// Mitsubishi GX Developer project: 20100302伺服締付機V02   PLC: FX3G

PROGRAM MAIN
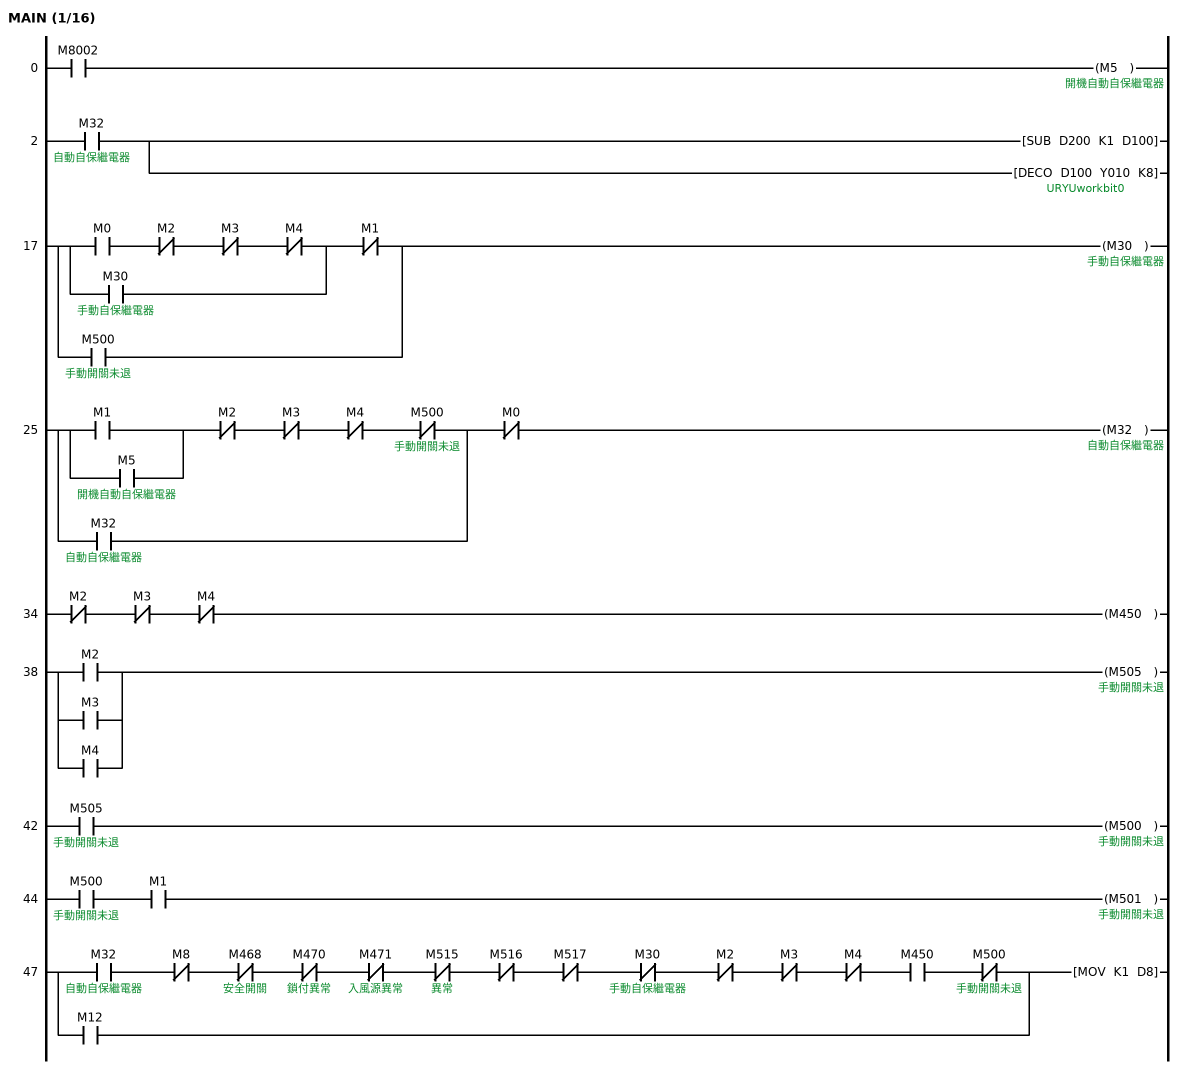
0     LD      M8002
      OUT     M5  ; 開機自動自保繼電器
2     LD      M32  ; 自動自保繼電器
      SUB     D200 K1 D100
        [note] 模組選擇
      DECO    D100 Y010 K8  ; URYUworkbit0
17    LD      M0
      ANI     M2
      ANI     M3
      ANI     M4
      OR      M30  ; 手動自保繼電器
      ANI     M1
      OR      M500  ; 手動開關未退
      OUT     M30  ; 手動自保繼電器
25    LD      M1
      OR      M5  ; 開機自動自保繼電器
      ANI     M2
      ANI     M3
      ANI     M4
      ANI     M500  ; 手動開關未退
      OR      M32  ; 自動自保繼電器
      ANI     M0
      OUT     M32  ; 自動自保繼電器
34    LDI     M2
      ANI     M3
      ANI     M4
      OUT     M450
38    LD      M2
      OR      M3
      OR      M4
      OUT     M505  ; 手動開關未退
42    LD      M505  ; 手動開關未退
      OUT     M500  ; 手動開關未退
44    LD      M500  ; 手動開關未退
      AND     M1
      OUT     M501  ; 手動開關未退
47    LD      M32  ; 自動自保繼電器
      ANI     M8
      ANI     M468  ; 安全開關
      ANI     M470  ; 鎖付異常
      ANI     M471  ; 入風源異常
      ANI     M515  ; 異常
      ANI     M516
      ANI     M517
      ANI     M30  ; 手動自保繼電器
      ANI     M2
      ANI     M3
      ANI     M4
      AND     M450
      ANI     M500  ; 手動開關未退
      OR      M12
      MOV     K1 D8
        [note] 自動畫面
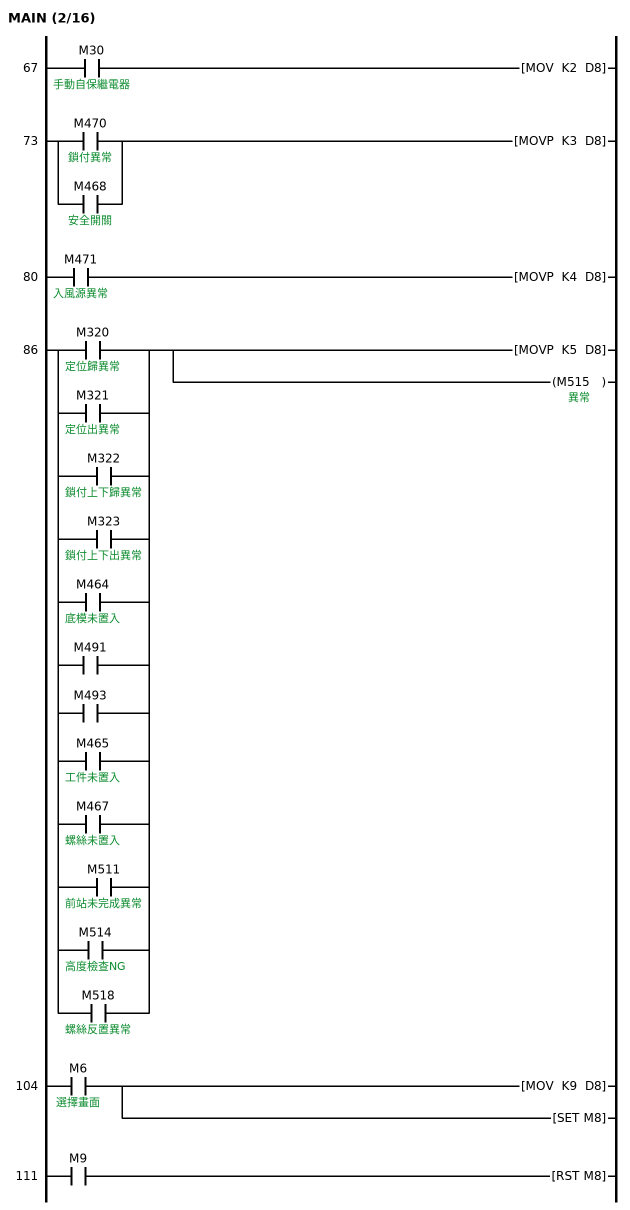
67    LD      M30  ; 手動自保繼電器
      MOV     K2 D8
        [note] 手動畫面
73    LD      M470  ; 鎖付異常
      OR      M468  ; 安全開關
      MOVP    K3 D8
        [note] 異常畫面
80    LD      M471  ; 入風源異常
      MOVP    K4 D8
        [note] 入風源異常畫面
86    LD      M320  ; 定位歸異常
      OR      M321  ; 定位出異常
      OR      M322  ; 鎖付上下歸異常
      OR      M323  ; 鎖付上下出異常
      OR      M464  ; 底模未置入
      OR      M491
      OR      M493
      OR      M465  ; 工件未置入
      OR      M467  ; 螺絲未置入
      OR      M511  ; 前站未完成異常
      OR      M514  ; 高度檢查NG
      OR      M518  ; 螺絲反置異常
      MOVP    K5 D8
        [note] 磁簧開關異常畫面
      OUT     M515  ; 異常
104   LD      M6  ; 選擇畫面
      MOV     K9 D8
      SET     M8
111   LD      M9
      RST     M8
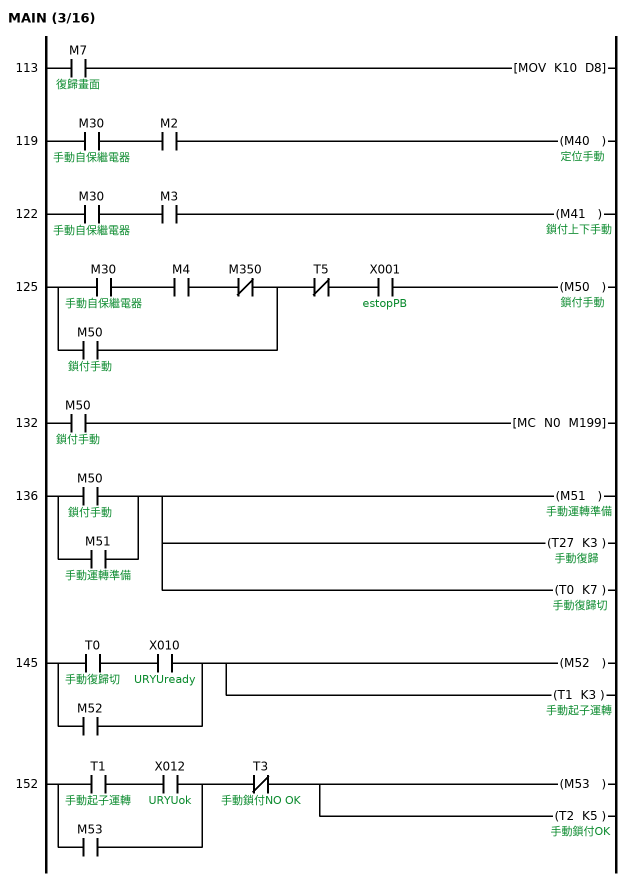
113   LD      M7  ; 復歸畫面
      MOV     K10 D8
119   LD      M30  ; 手動自保繼電器
      AND     M2
      OUT     M40  ; 定位手動
122   LD      M30  ; 手動自保繼電器
      AND     M3
      OUT     M41  ; 鎖付上下手動
125   LD      M30  ; 手動自保繼電器
      AND     M4
      ANI     M350
      OR      M50  ; 鎖付手動
      ANI     T5
      AND     X001  ; estopPB
      OUT     M50  ; 鎖付手動
132   LD      M50  ; 鎖付手動
      MC      N0 M199
136   LD      M50  ; 鎖付手動
      OR      M51  ; 手動運轉準備
      OUT     M51  ; 手動運轉準備
      OUT     T27 K3  ; 手動復歸
      OUT     T0 K7  ; 手動復歸切
145   LD      T0  ; 手動復歸切
      AND     X010  ; URYUready
      OR      M52
      OUT     M52
      OUT     T1 K3  ; 手動起子運轉
152   LD      T1  ; 手動起子運轉
      AND     X012  ; URYUok
      OR      M53
      ANI     T3  ; 手動鎖付NO OK
      OUT     M53
      OUT     T2 K5  ; 手動鎖付OK
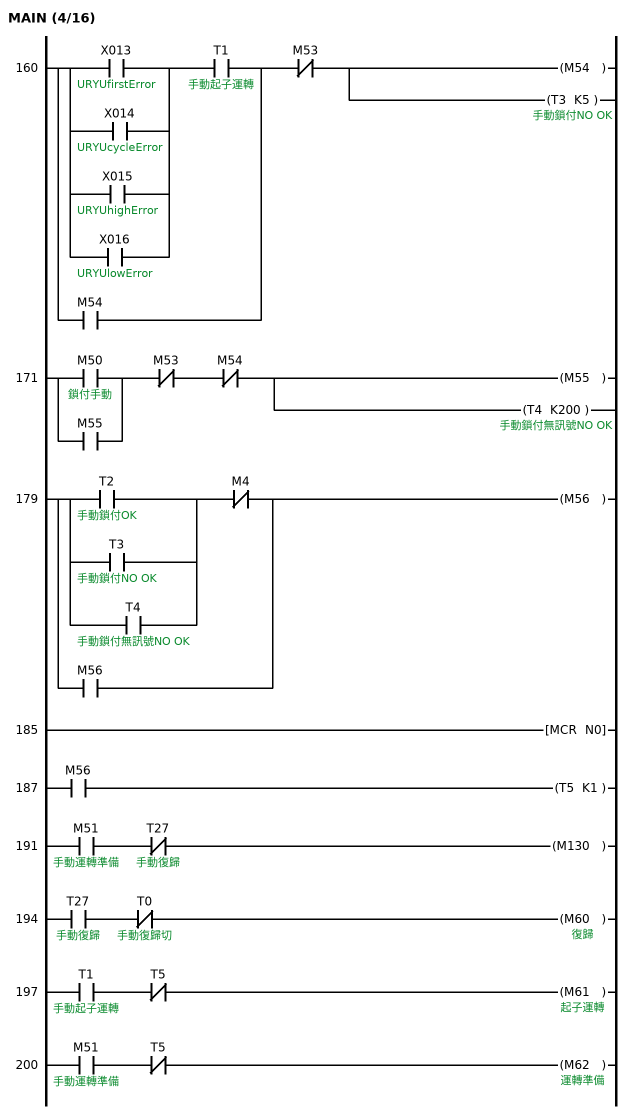
160   LD      X013  ; URYUfirstError
      OR      X014  ; URYUcycleError
      OR      X015  ; URYUhighError
      OR      X016  ; URYUlowError
      AND     T1  ; 手動起子運轉
      OR      M54
      ANI     M53
      OUT     M54
      OUT     T3 K5  ; 手動鎖付NO OK
171   LD      M50  ; 鎖付手動
      OR      M55
      ANI     M53
      ANI     M54
      OUT     M55
      OUT     T4 K200  ; 手動鎖付無訊號NO OK
179   LD      T2  ; 手動鎖付OK
      OR      T3  ; 手動鎖付NO OK
      OR      T4  ; 手動鎖付無訊號NO OK
      ANI     M4
      OR      M56
      OUT     M56
185   MCR     N0
187   LD      M56
      OUT     T5 K1
191   LD      M51  ; 手動運轉準備
      ANI     T27  ; 手動復歸
      OUT     M130
194   LD      T27  ; 手動復歸
      ANI     T0  ; 手動復歸切
      OUT     M60  ; 復歸
197   LD      T1  ; 手動起子運轉
      ANI     T5
      OUT     M61  ; 起子運轉
200   LD      M51  ; 手動運轉準備
      ANI     T5
      OUT     M62  ; 運轉準備
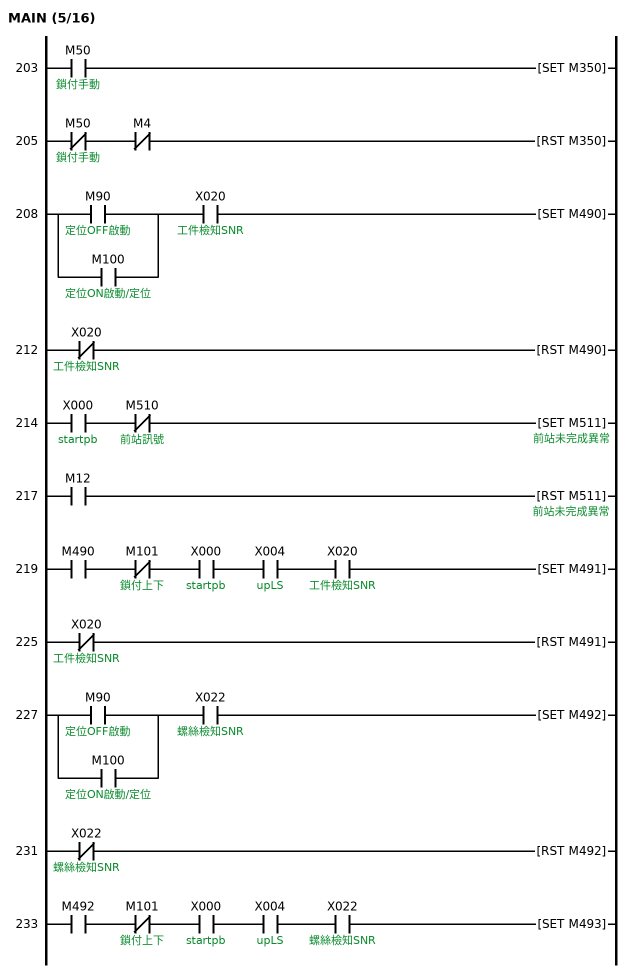
203   LD      M50  ; 鎖付手動
      SET     M350
205   LDI     M50  ; 鎖付手動
      ANI     M4
      RST     M350
208   LD      M90  ; 定位OFF啟動
      OR      M100  ; 定位ON啟動/定位
      AND     X020  ; 工件檢知SNR
      SET     M490
212   LDI     X020  ; 工件檢知SNR
      RST     M490
214   LD      X000  ; startpb
      ANI     M510  ; 前站訊號
      SET     M511  ; 前站未完成異常
217   LD      M12
      RST     M511  ; 前站未完成異常
219   LD      M490
      ANI     M101  ; 鎖付上下
      AND     X000  ; startpb
      AND     X004  ; upLS
      AND     X020  ; 工件檢知SNR
      SET     M491
225   LDI     X020  ; 工件檢知SNR
      RST     M491
227   LD      M90  ; 定位OFF啟動
      OR      M100  ; 定位ON啟動/定位
      AND     X022  ; 螺絲檢知SNR
      SET     M492
231   LDI     X022  ; 螺絲檢知SNR
      RST     M492
233   LD      M492
      ANI     M101  ; 鎖付上下
      AND     X000  ; startpb
      AND     X004  ; upLS
      AND     X022  ; 螺絲檢知SNR
      SET     M493
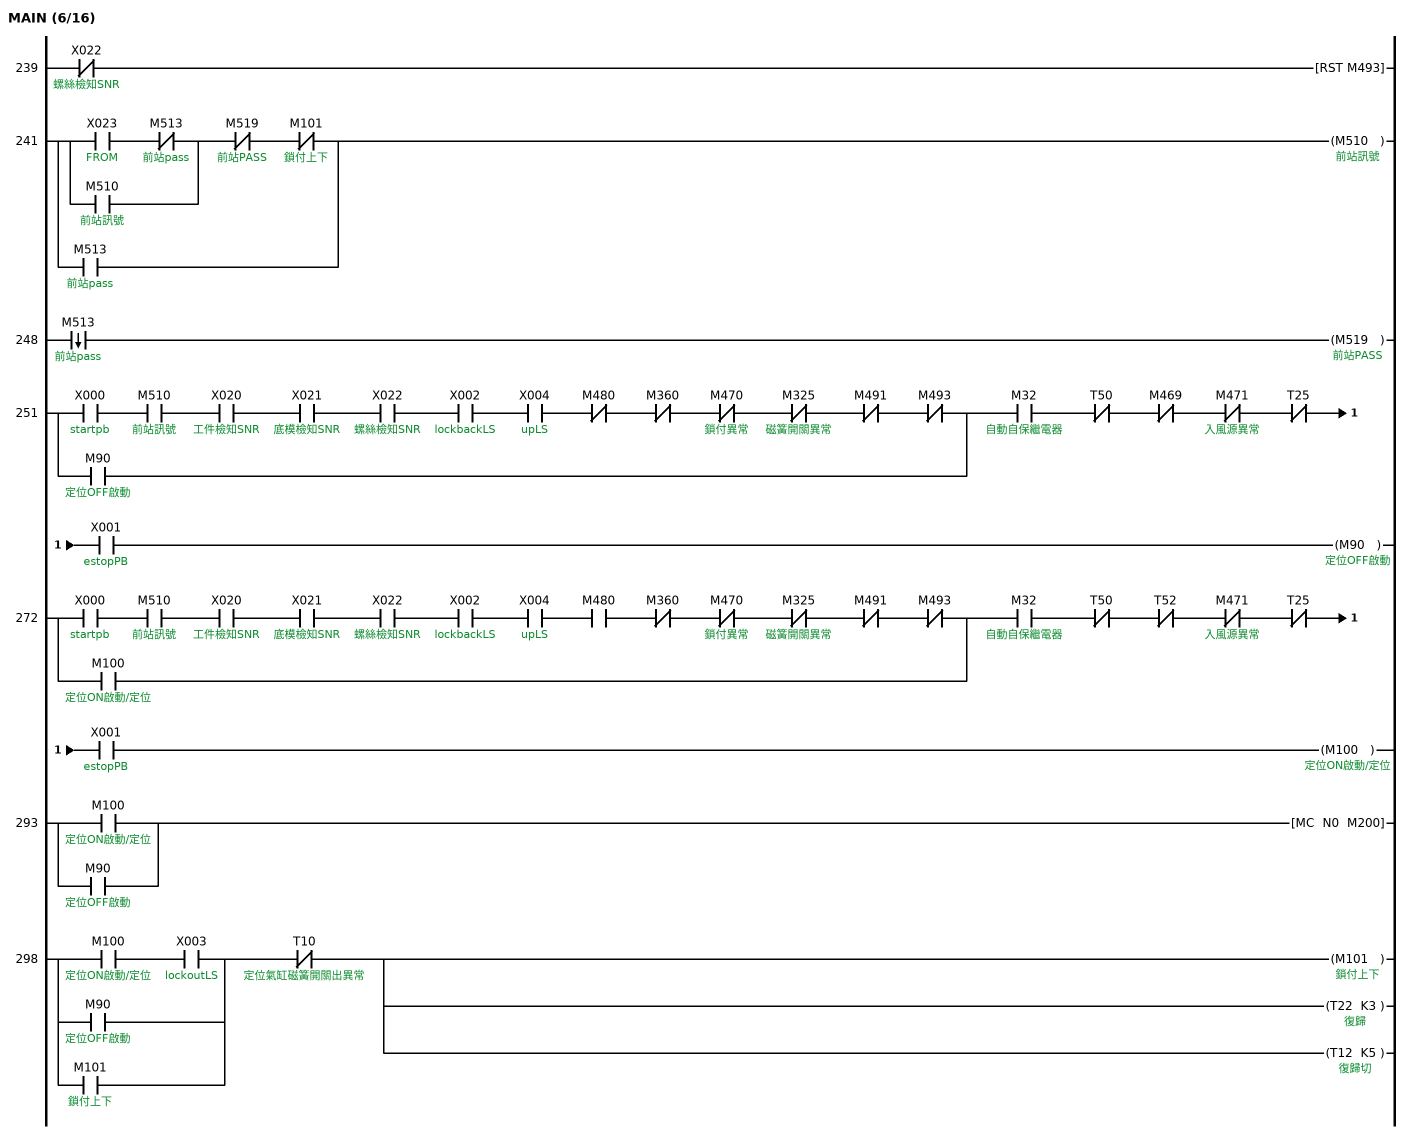
239   LDI     X022  ; 螺絲檢知SNR
      RST     M493
241   LD      X023  ; FROM
      ANI     M513  ; 前站pass
      OR      M510  ; 前站訊號
      ANI     M519  ; 前站PASS
      ANI     M101  ; 鎖付上下
      OR      M513  ; 前站pass
      OUT     M510  ; 前站訊號
248   LDF     M513  ; 前站pass
      OUT     M519  ; 前站PASS
251   LD      X000  ; startpb
      AND     M510  ; 前站訊號
      AND     X020  ; 工件檢知SNR
      AND     X021  ; 底模檢知SNR
      AND     X022  ; 螺絲檢知SNR
      AND     X002  ; lockbackLS
      AND     X004  ; upLS
      ANI     M480
      ANI     M360
      ANI     M470  ; 鎖付異常
      ANI     M325  ; 磁簧開關異常
      ANI     M491
      ANI     M493
      OR      M90  ; 定位OFF啟動
      AND     M32  ; 自動自保繼電器
      ANI     T50
      ANI     M469
      ANI     M471  ; 入風源異常
      ANI     T25
      AND     X001  ; estopPB
      OUT     M90  ; 定位OFF啟動
272   LD      X000  ; startpb
      AND     M510  ; 前站訊號
      AND     X020  ; 工件檢知SNR
      AND     X021  ; 底模檢知SNR
      AND     X022  ; 螺絲檢知SNR
      AND     X002  ; lockbackLS
      AND     X004  ; upLS
      AND     M480
      ANI     M360
      ANI     M470  ; 鎖付異常
      ANI     M325  ; 磁簧開關異常
      ANI     M491
      ANI     M493
      OR      M100  ; 定位ON啟動/定位
      AND     M32  ; 自動自保繼電器
      ANI     T50
      ANI     T52
      ANI     M471  ; 入風源異常
      ANI     T25
      AND     X001  ; estopPB
      OUT     M100  ; 定位ON啟動/定位
293   LD      M100  ; 定位ON啟動/定位
      OR      M90  ; 定位OFF啟動
      MC      N0 M200
298   LD      M100  ; 定位ON啟動/定位
      AND     X003  ; lockoutLS
      OR      M90  ; 定位OFF啟動
      OR      M101  ; 鎖付上下
      ANI     T10  ; 定位氣缸磁簧開關出異常
      OUT     M101  ; 鎖付上下
      OUT     T22 K3  ; 復歸
      OUT     T12 K5  ; 復歸切
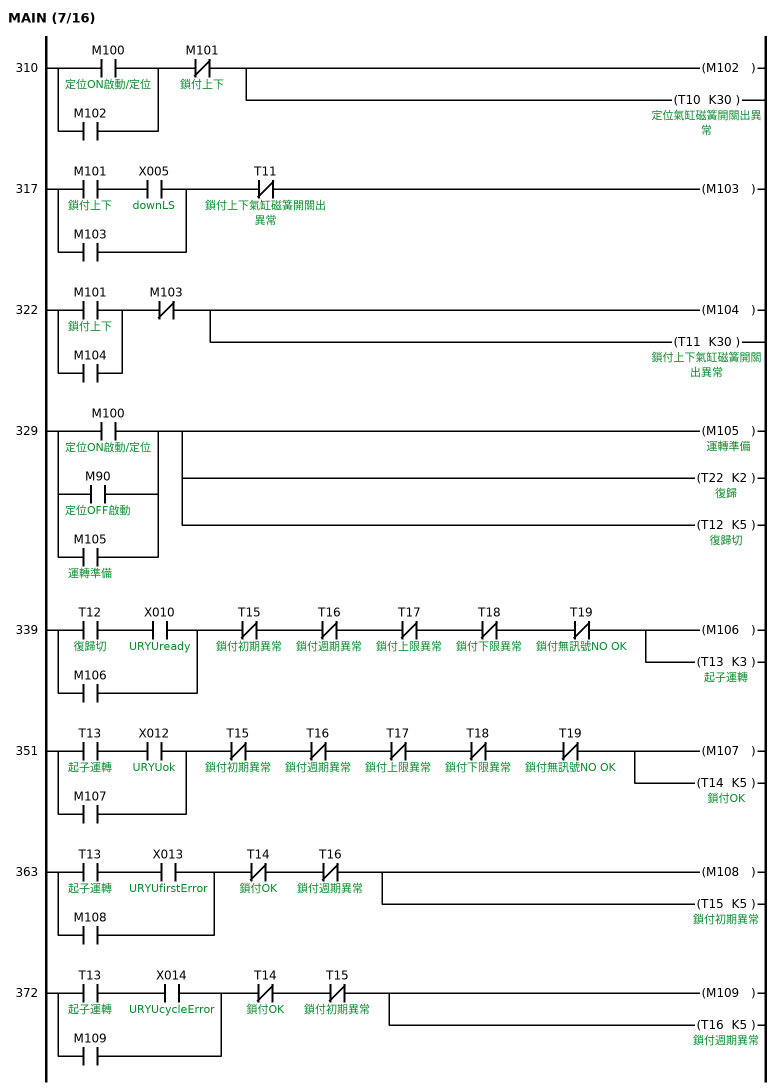
310   LD      M100  ; 定位ON啟動/定位
      OR      M102
      ANI     M101  ; 鎖付上下
      OUT     M102
      OUT     T10 K30  ; 定位氣缸磁簧開關出異常
317   LD      M101  ; 鎖付上下
      AND     X005  ; downLS
      OR      M103
      ANI     T11  ; 鎖付上下氣缸磁簧開關出異常
      OUT     M103
322   LD      M101  ; 鎖付上下
      OR      M104
      ANI     M103
      OUT     M104
      OUT     T11 K30  ; 鎖付上下氣缸磁簧開關出異常
329   LD      M100  ; 定位ON啟動/定位
      OR      M90  ; 定位OFF啟動
      OR      M105  ; 運轉準備
      OUT     M105  ; 運轉準備
      OUT     T22 K2  ; 復歸
      OUT     T12 K5  ; 復歸切
339   LD      T12  ; 復歸切
      AND     X010  ; URYUready
      OR      M106
      ANI     T15  ; 鎖付初期異常
      ANI     T16  ; 鎖付週期異常
      ANI     T17  ; 鎖付上限異常
      ANI     T18  ; 鎖付下限異常
      ANI     T19  ; 鎖付無訊號NO OK
      OUT     M106
      OUT     T13 K3  ; 起子運轉
351   LD      T13  ; 起子運轉
      AND     X012  ; URYUok
      OR      M107
      ANI     T15  ; 鎖付初期異常
      ANI     T16  ; 鎖付週期異常
      ANI     T17  ; 鎖付上限異常
      ANI     T18  ; 鎖付下限異常
      ANI     T19  ; 鎖付無訊號NO OK
      OUT     M107
      OUT     T14 K5  ; 鎖付OK
363   LD      T13  ; 起子運轉
      AND     X013  ; URYUfirstError
      OR      M108
      ANI     T14  ; 鎖付OK
      ANI     T16  ; 鎖付週期異常
      OUT     M108
      OUT     T15 K5  ; 鎖付初期異常
372   LD      T13  ; 起子運轉
      AND     X014  ; URYUcycleError
      OR      M109
      ANI     T14  ; 鎖付OK
      ANI     T15  ; 鎖付初期異常
      OUT     M109
      OUT     T16 K5  ; 鎖付週期異常
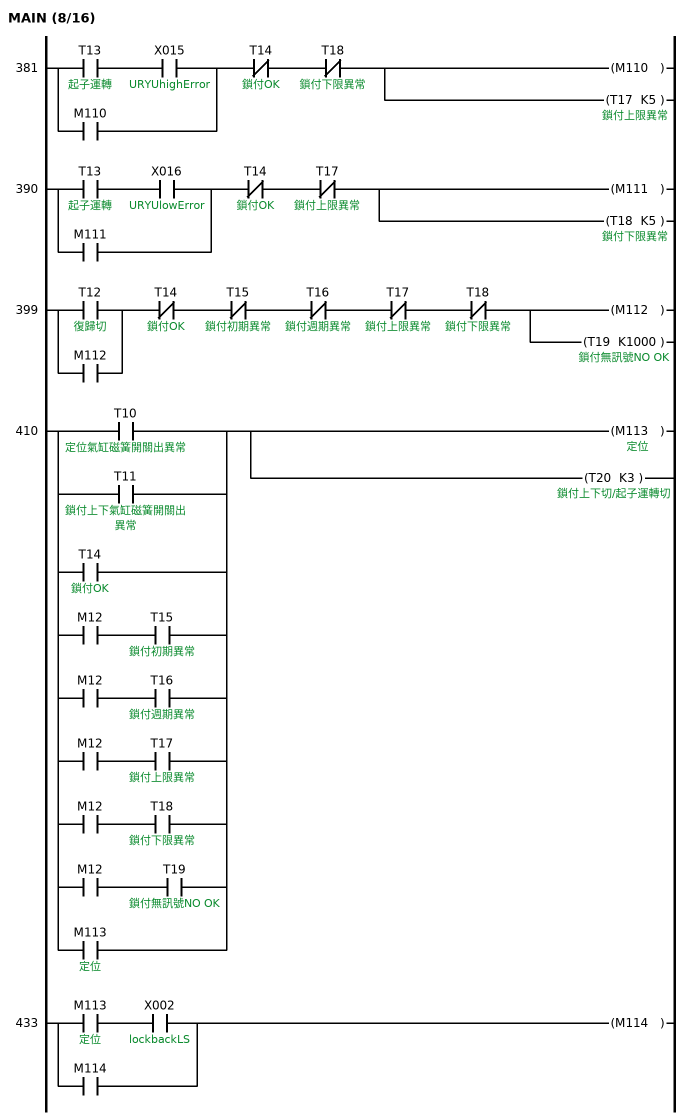
381   LD      T13  ; 起子運轉
      AND     X015  ; URYUhighError
      OR      M110
      ANI     T14  ; 鎖付OK
      ANI     T18  ; 鎖付下限異常
      OUT     M110
      OUT     T17 K5  ; 鎖付上限異常
390   LD      T13  ; 起子運轉
      AND     X016  ; URYUlowError
      OR      M111
      ANI     T14  ; 鎖付OK
      ANI     T17  ; 鎖付上限異常
      OUT     M111
      OUT     T18 K5  ; 鎖付下限異常
399   LD      T12  ; 復歸切
      OR      M112
      ANI     T14  ; 鎖付OK
      ANI     T15  ; 鎖付初期異常
      ANI     T16  ; 鎖付週期異常
      ANI     T17  ; 鎖付上限異常
      ANI     T18  ; 鎖付下限異常
      OUT     M112
      OUT     T19 K1000  ; 鎖付無訊號NO OK
410   LD      T10  ; 定位氣缸磁簧開關出異常
      OR      T11  ; 鎖付上下氣缸磁簧開關出異常
      OR      T14  ; 鎖付OK
      LD      M12
      AND     T15  ; 鎖付初期異常
      ORB
      LD      M12
      AND     T16  ; 鎖付週期異常
      ORB
      LD      M12
      AND     T17  ; 鎖付上限異常
      ORB
      LD      M12
      AND     T18  ; 鎖付下限異常
      ORB
      LD      M12
      AND     T19  ; 鎖付無訊號NO OK
      ORB
      OR      M113  ; 定位
      OUT     M113  ; 定位
      OUT     T20 K3  ; 鎖付上下切/起子運轉切
433   LD      M113  ; 定位
      AND     X002  ; lockbackLS
      OR      M114
      OUT     M114
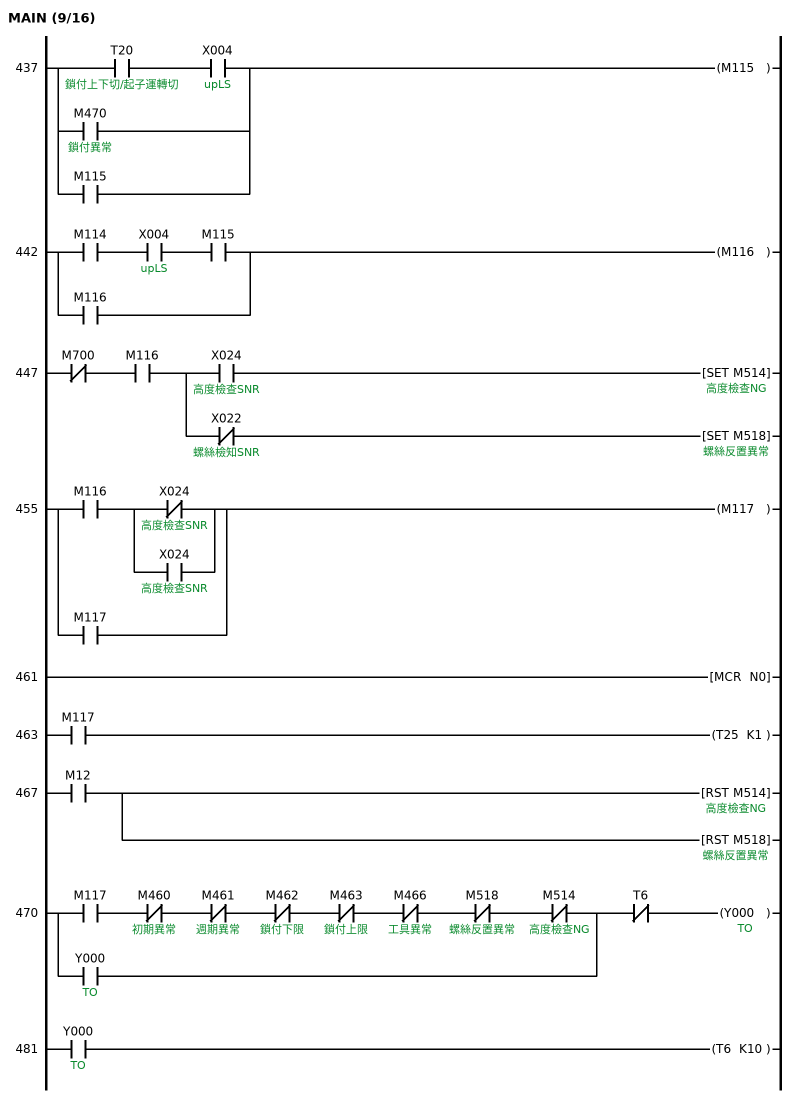
437   LD      T20  ; 鎖付上下切/起子運轉切
      AND     X004  ; upLS
      OR      M470  ; 鎖付異常
      OR      M115
      OUT     M115
442   LD      M114
      AND     X004  ; upLS
      AND     M115
      OR      M116
      OUT     M116
447   LDI     M700
      AND     M116
      MPS
      AND     X024  ; 高度檢查SNR
      SET     M514  ; 高度檢查NG
      MPP
      ANI     X022  ; 螺絲檢知SNR
      SET     M518  ; 螺絲反置異常
455   LD      M116
      LDI     X024  ; 高度檢查SNR
      OR      X024  ; 高度檢查SNR
      ANB
      OR      M117
      OUT     M117
461   MCR     N0
463   LD      M117
      OUT     T25 K1
467   LD      M12
      RST     M514  ; 高度檢查NG
      RST     M518  ; 螺絲反置異常
470   LD      M117
      ANI     M460  ; 初期異常
      ANI     M461  ; 週期異常
      ANI     M462  ; 鎖付下限
      ANI     M463  ; 鎖付上限
      ANI     M466  ; 工具異常
      ANI     M518  ; 螺絲反置異常
      ANI     M514  ; 高度檢查NG
      OR      Y000  ; TO
      ANI     T6
      OUT     Y000  ; TO
481   LD      Y000  ; TO
      OUT     T6 K10
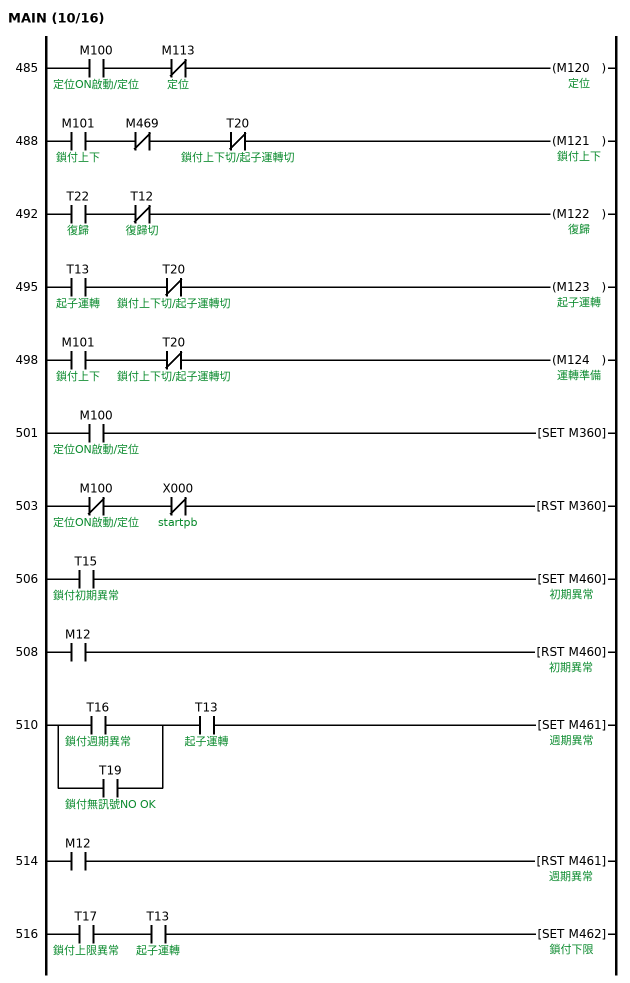
485   LD      M100  ; 定位ON啟動/定位
      ANI     M113  ; 定位
      OUT     M120  ; 定位
488   LD      M101  ; 鎖付上下
      ANI     M469
      ANI     T20  ; 鎖付上下切/起子運轉切
      OUT     M121  ; 鎖付上下
492   LD      T22  ; 復歸
      ANI     T12  ; 復歸切
      OUT     M122  ; 復歸
495   LD      T13  ; 起子運轉
      ANI     T20  ; 鎖付上下切/起子運轉切
      OUT     M123  ; 起子運轉
498   LD      M101  ; 鎖付上下
      ANI     T20  ; 鎖付上下切/起子運轉切
      OUT     M124  ; 運轉準備
501   LD      M100  ; 定位ON啟動/定位
      SET     M360
503   LDI     M100  ; 定位ON啟動/定位
      ANI     X000  ; startpb
      RST     M360
506   LD      T15  ; 鎖付初期異常
      SET     M460  ; 初期異常
508   LD      M12
      RST     M460  ; 初期異常
510   LD      T16  ; 鎖付週期異常
      OR      T19  ; 鎖付無訊號NO OK
      AND     T13  ; 起子運轉
      SET     M461  ; 週期異常
514   LD      M12
      RST     M461  ; 週期異常
516   LD      T17  ; 鎖付上限異常
      AND     T13  ; 起子運轉
      SET     M462  ; 鎖付下限
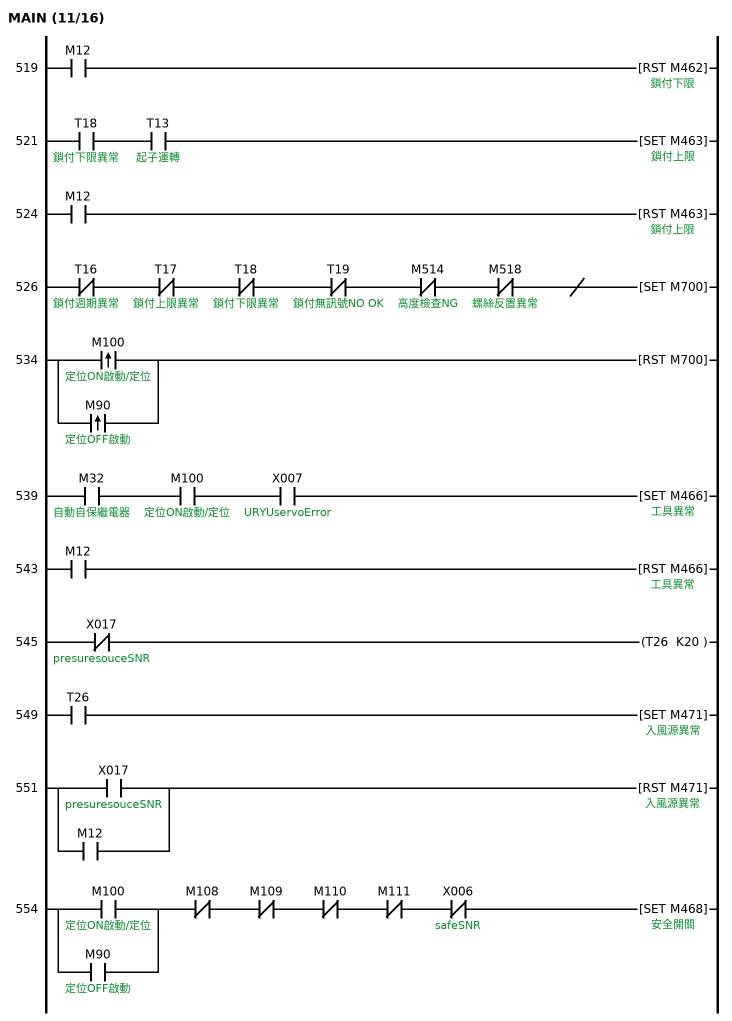
519   LD      M12
      RST     M462  ; 鎖付下限
521   LD      T18  ; 鎖付下限異常
      AND     T13  ; 起子運轉
      SET     M463  ; 鎖付上限
524   LD      M12
      RST     M463  ; 鎖付上限
526   LDI     T16  ; 鎖付週期異常
      ANI     T17  ; 鎖付上限異常
      ANI     T18  ; 鎖付下限異常
      ANI     T19  ; 鎖付無訊號NO OK
      ANI     M514  ; 高度檢查NG
      ANI     M518  ; 螺絲反置異常
      INV
      SET     M700
534   LDP     M100  ; 定位ON啟動/定位
      ORP     M90  ; 定位OFF啟動
      RST     M700
539   LD      M32  ; 自動自保繼電器
      AND     M100  ; 定位ON啟動/定位
      AND     X007  ; URYUservoError
      SET     M466  ; 工具異常
543   LD      M12
      RST     M466  ; 工具異常
545   LDI     X017  ; presuresouceSNR
      OUT     T26 K20
549   LD      T26
      SET     M471  ; 入風源異常
551   LD      X017  ; presuresouceSNR
      OR      M12
      RST     M471  ; 入風源異常
554   LD      M100  ; 定位ON啟動/定位
      OR      M90  ; 定位OFF啟動
      ANI     M108
      ANI     M109
      ANI     M110
      ANI     M111
      ANI     X006  ; safeSNR
      SET     M468  ; 安全開關
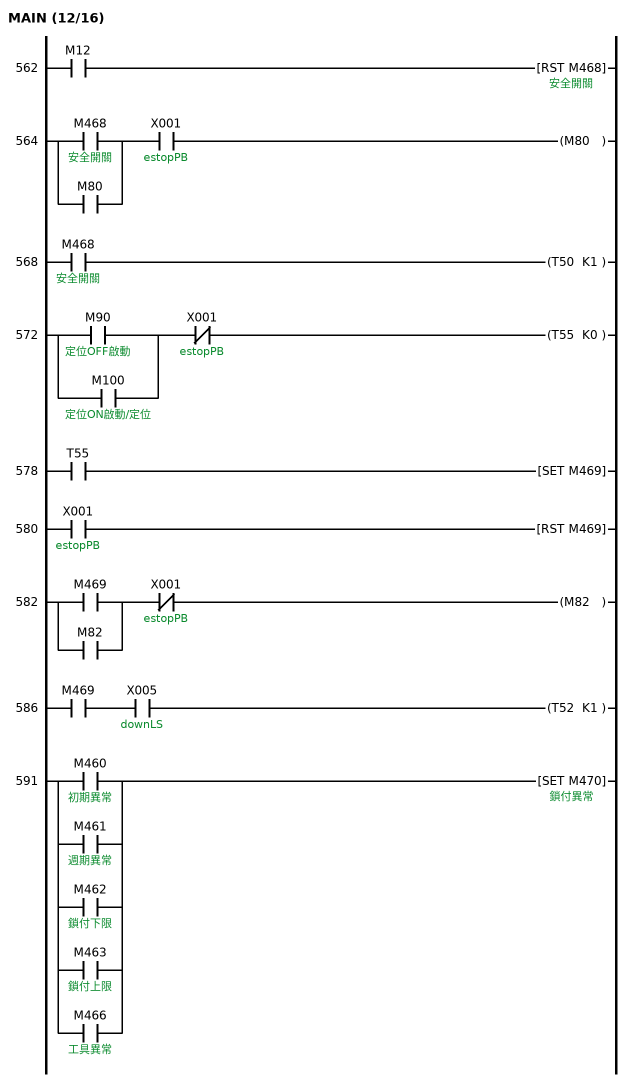
562   LD      M12
      RST     M468  ; 安全開關
564   LD      M468  ; 安全開關
      OR      M80
      AND     X001  ; estopPB
      OUT     M80
568   LD      M468  ; 安全開關
      OUT     T50 K1
572   LD      M90  ; 定位OFF啟動
      OR      M100  ; 定位ON啟動/定位
      ANI     X001  ; estopPB
      OUT     T55 K0
578   LD      T55
      SET     M469
580   LD      X001  ; estopPB
      RST     M469
582   LD      M469
      OR      M82
      ANI     X001  ; estopPB
      OUT     M82
586   LD      M469
      AND     X005  ; downLS
      OUT     T52 K1
591   LD      M460  ; 初期異常
      OR      M461  ; 週期異常
      OR      M462  ; 鎖付下限
      OR      M463  ; 鎖付上限
      OR      M466  ; 工具異常
      SET     M470  ; 鎖付異常
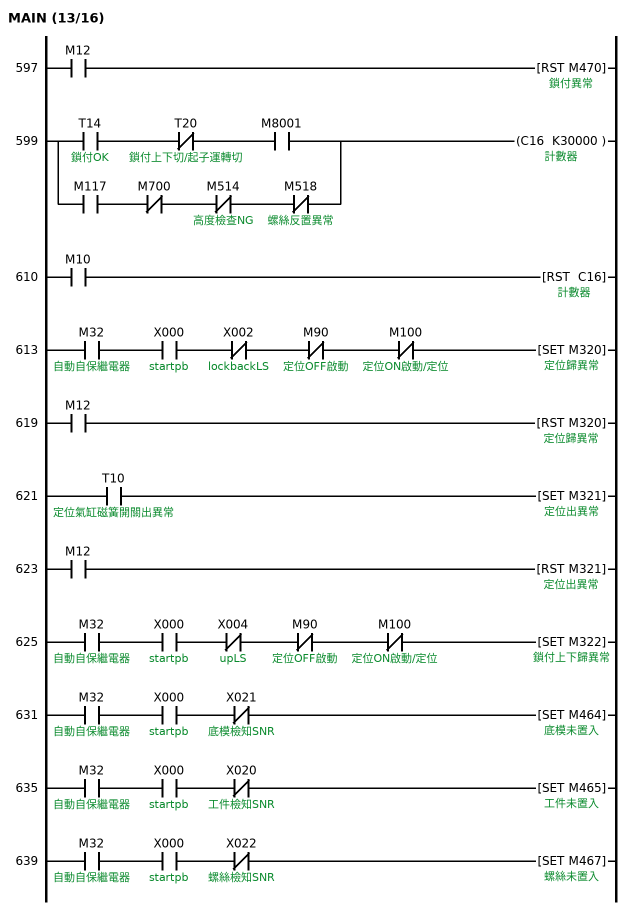
597   LD      M12
      RST     M470  ; 鎖付異常
599   LD      T14  ; 鎖付OK
      ANI     T20  ; 鎖付上下切/起子運轉切
      AND     M8001
      LD      M117
      ANI     M700
      ANI     M514  ; 高度檢查NG
      ANI     M518  ; 螺絲反置異常
      ORB
      OUT     C16 K30000  ; 計數器
610   LD      M10
      RST     C16  ; 計數器
613   LD      M32  ; 自動自保繼電器
      AND     X000  ; startpb
      ANI     X002  ; lockbackLS
      ANI     M90  ; 定位OFF啟動
      ANI     M100  ; 定位ON啟動/定位
      SET     M320  ; 定位歸異常
619   LD      M12
      RST     M320  ; 定位歸異常
621   LD      T10  ; 定位氣缸磁簧開關出異常
      SET     M321  ; 定位出異常
623   LD      M12
      RST     M321  ; 定位出異常
625   LD      M32  ; 自動自保繼電器
      AND     X000  ; startpb
      ANI     X004  ; upLS
      ANI     M90  ; 定位OFF啟動
      ANI     M100  ; 定位ON啟動/定位
      SET     M322  ; 鎖付上下歸異常
631   LD      M32  ; 自動自保繼電器
      AND     X000  ; startpb
      ANI     X021  ; 底模檢知SNR
      SET     M464  ; 底模未置入
635   LD      M32  ; 自動自保繼電器
      AND     X000  ; startpb
      ANI     X020  ; 工件檢知SNR
      SET     M465  ; 工件未置入
639   LD      M32  ; 自動自保繼電器
      AND     X000  ; startpb
      ANI     X022  ; 螺絲檢知SNR
      SET     M467  ; 螺絲未置入
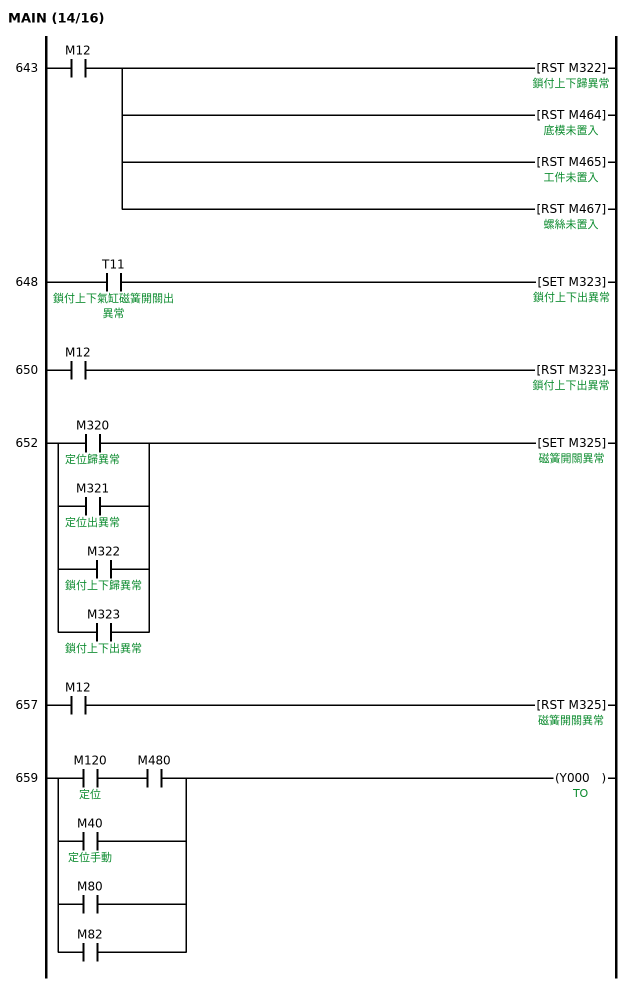
643   LD      M12
      RST     M322  ; 鎖付上下歸異常
      RST     M464  ; 底模未置入
      RST     M465  ; 工件未置入
      RST     M467  ; 螺絲未置入
648   LD      T11  ; 鎖付上下氣缸磁簧開關出異常
      SET     M323  ; 鎖付上下出異常
650   LD      M12
      RST     M323  ; 鎖付上下出異常
652   LD      M320  ; 定位歸異常
      OR      M321  ; 定位出異常
      OR      M322  ; 鎖付上下歸異常
      OR      M323  ; 鎖付上下出異常
      SET     M325  ; 磁簧開關異常
657   LD      M12
      RST     M325  ; 磁簧開關異常
659   LD      M120  ; 定位
      AND     M480
      OR      M40  ; 定位手動
      OR      M80
      OR      M82
      OUT     Y000  ; TO
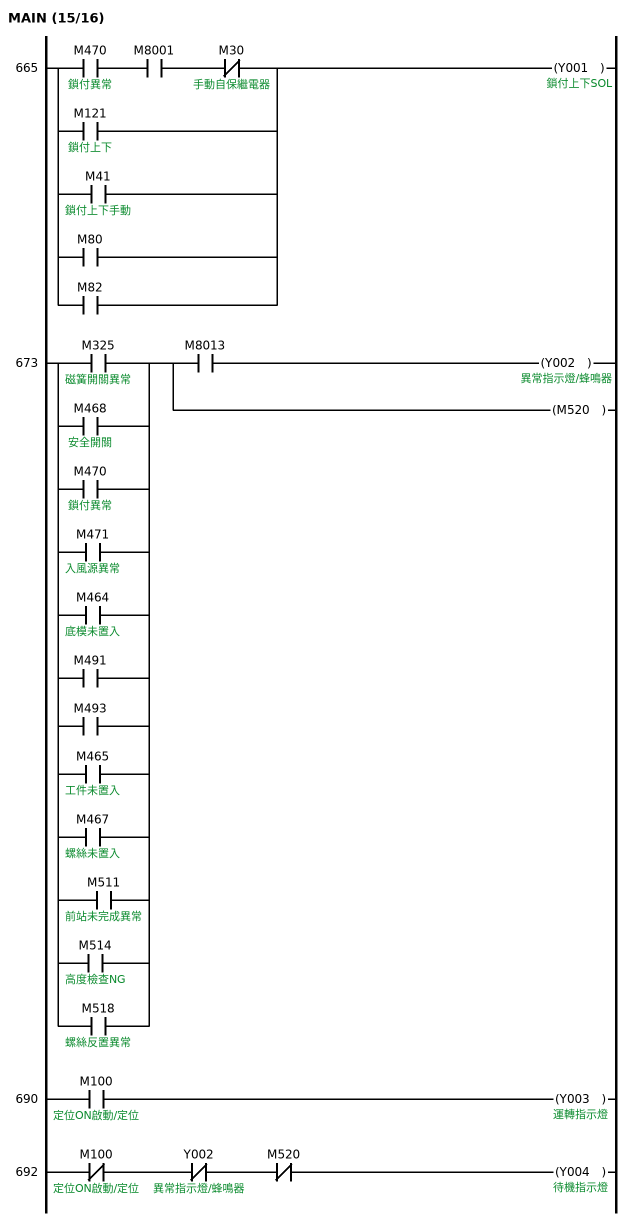
665   LD      M470  ; 鎖付異常
      AND     M8001
      ANI     M30  ; 手動自保繼電器
      OR      M121  ; 鎖付上下
      OR      M41  ; 鎖付上下手動
      OR      M80
      OR      M82
      OUT     Y001  ; 鎖付上下SOL
673   LD      M325  ; 磁簧開關異常
      OR      M468  ; 安全開關
      OR      M470  ; 鎖付異常
      OR      M471  ; 入風源異常
      OR      M464  ; 底模未置入
      OR      M491
      OR      M493
      OR      M465  ; 工件未置入
      OR      M467  ; 螺絲未置入
      OR      M511  ; 前站未完成異常
      OR      M514  ; 高度檢查NG
      OR      M518  ; 螺絲反置異常
      MPS
      AND     M8013
      OUT     Y002  ; 異常指示燈/蜂鳴器
      MPP
      OUT     M520
690   LD      M100  ; 定位ON啟動/定位
      OUT     Y003  ; 運轉指示燈
692   LDI     M100  ; 定位ON啟動/定位
      ANI     Y002  ; 異常指示燈/蜂鳴器
      ANI     M520
      OUT     Y004  ; 待機指示燈
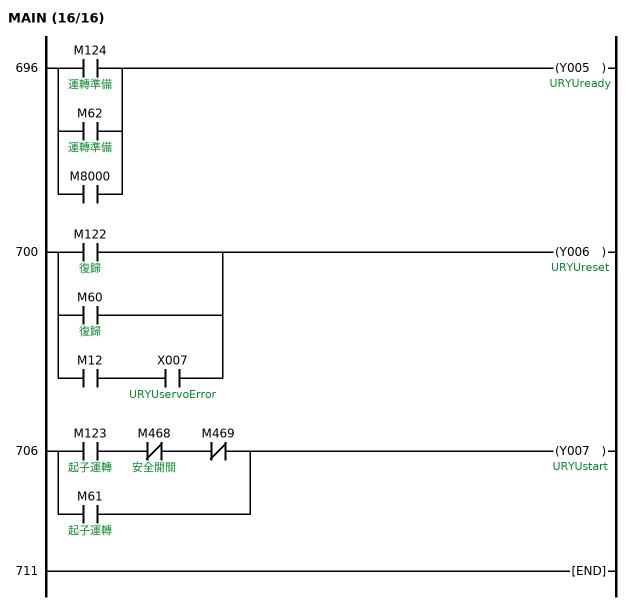
696   LD      M124  ; 運轉準備
      OR      M62  ; 運轉準備
      OR      M8000
      OUT     Y005  ; URYUready
700   LD      M122  ; 復歸
      OR      M60  ; 復歸
      LD      M12
      AND     X007  ; URYUservoError
      ORB
      OUT     Y006  ; URYUreset
706   LD      M123  ; 起子運轉
      ANI     M468  ; 安全開關
      ANI     M469
      OR      M61  ; 起子運轉
      OUT     Y007  ; URYUstart
711   END
END_PROGRAM

// device comments not shown above
X011  ; URYUcomplite
Y011  ; URYUworkbit1
Y012  ; URYUworkbit2
Y013  ; URYUworkbit3
Y014  ; URYUworkbit4
Y015  ; URYUworkbit5
Y016  ; URYUworkbit6
Y017  ; URYUworkbit7
